{attribute 'GeneratedUsingTerminal: EL2014-0000-0016'}
{attribute addProperty BoxType "EL2014-0000-0016"}
{attribute addProperty Id "OutputBOOL1"}
{attribute addProperty CRC "3592680812"}
{attribute addProperty Size "1"}
TYPE Channel_D623F56C :
STRUCT
	{attribute addProperty Name "Output"}
	Output : BOOL;
END_STRUCT
END_TYPE

(* stored: Version 1.2.0.0, ProductVersion 3.1.4024.11
   DUT Channel_D623F56C: Id {d36a1233-7f99-477f-b83d-28d1a1af92f6} *)
